// TIA Portal V19 export
DATA_BLOCK "Setpoints"   // DB111
{ S7_Optimized_Access := 'TRUE' }
VERSION : 0.0
// stored: AutoNumber false, MemoryReserve 0
   VAR RETAIN
      TT0176MinTempUnster : Real := 125.0;   // MIN. TEMPERATUR TT 01.76 = UNSTERILE
      TT0160MinTempUnster : Real := 125.0;   // MIN. TEMPERATUR TT 01.60 = UNSTERILE
      TT0163MinTempUnster : Real := 125.0;   // MIN. TEMPERATUR TT 01.63 = UNSTERILE
      TT0178MinTempUnster : Real := 125.0;   // MIN. TEMPERATUR TT 01.78 = UNSTERILE
      TT0176LowTemp : Real := 110.0;   // ALARM TEMPERATUR TT 01.76 LOW
      TT0178LowTemp : Real := 110.0;   // ALARM TEMPERATUR TT 01.78 LOW
      TT0176StartSterileTime : Real := 126.0;   // START STERILETIME TT 01.76
      TT0160StartSterileTime : Real := 126.0;   // START STERILETIME TT 01.60
      TT0163StartSterileTime : Real := 126.0;   // START STERILETIME TT 01.63
      TT0178StartSterileTime : Real := 126.0;   // START STERILETIME TT 01.78
      TT0176MaxTotalStop : Real := 100.0;   // MAX TEMPERATUR TT 01.76 FOR TOTAL STOP
      PresForOpenDrain : Real := 500.0;   // OPEN DRAIN AT COOLING IF PRESSURE TOO LOW
      TT01172SpLyeFiller : Real := 75.0;   // SETPOINT DURING LYECIRCULATION FILLER
      TT01172SpAcidFiller : Real := 60.0;   // SETPOINT DURING ACID CIRCULATION FILLER
      TT0172SpLye : Real := 75.0;   // SETPOINT DURING LYE CIRCULATION
      TT0172SpAcid : Real := 59.0;   // SETPOINT DURING ACID CIRCULATION
      MinCipReturTempTT01 : Real := 50.0;   // MIN.TEMP.BEFORE START CIRC. TIMER
      MinCipFillerTempTT01 : Real := 55.0;   // MIN.TEMP.BEFORE START CIRC. TIMER FILLER
      PT0167StopCooling : Real := 1.0;   // STOP COOLING AT PT 01.67
      PT0167RestartCooling : Real := 1.1;   // RESTART COOLING AT PT 01.67
      StartBlowOutMinPressure : Real := 0.7;   // MIN. PRESS FOR START BLOW OUT
      PT0167SpProduction : Real := 2.5;   // FILLING PRESSURE IN PRODUCTION
      PT0167SpCIP : Real := 1.3;   // PRESSURE DURING CIP
      PT0167SpInCooling : Real := 1.8;   // SETPOINT PRESSURE DURING COOLING
      StartCipMinPressure : Real := 0.7;   // MIN.PRESSURE BEFORE START CIP
      MinPresUnsterile : Real := 0.3;   // MIN PRESSURE BEFORE UNSTERILE
      PT0167LowPressure : Real := 0.5;   // ALARM LOW PRESSURE PT 01.67
      StaPulseY0113 : Real := 98.0;   // START PULSING 01.13 AT TT 01.76=
      CloseY0113 : Real := 95.0;   // STOP PULSING 01.13 AT TT 01.76=
      OpenY0113AtLowTemp : Real := 90.0;   // OPEN 01.13 AT LOW TEMPERATURE
      CT2073LyeConcSpCIP : Real := 40.0;   // SETPOINT LYE CONCENTRATION
      CT2073AcidConcSpCIP : Real := 7.0;   // SETPOINT ACID CONCENTRATION
      CT2073MaxDeviationConcSp : Real := 1.0;   // DEVIATION FROM CONCENTRATION SETPOINT IN PERCENT
      PT0167SpCIPLow : Real := 0.8;
      ProgCIPFiller : Int;   // CIP PROGRAM FILLER
      ChainWashTempSetp : Real := 70.0;   // CHAIN WASH TEMPERATURE SETPOINT
      CT2073LyeConcSpFiller : Real := 20.0;
      CT2073AcidConcSpFiller : Real := 7.0;
      PT0167AcidPressure : Real := 0.6;
      TT0172SpPrerinse : Real := 35.0;   // Pre-rinse temperature SP
   END_VAR
BEGIN
END_DATA_BLOCK
